RoboDK station: robodk_dot_following.rdk

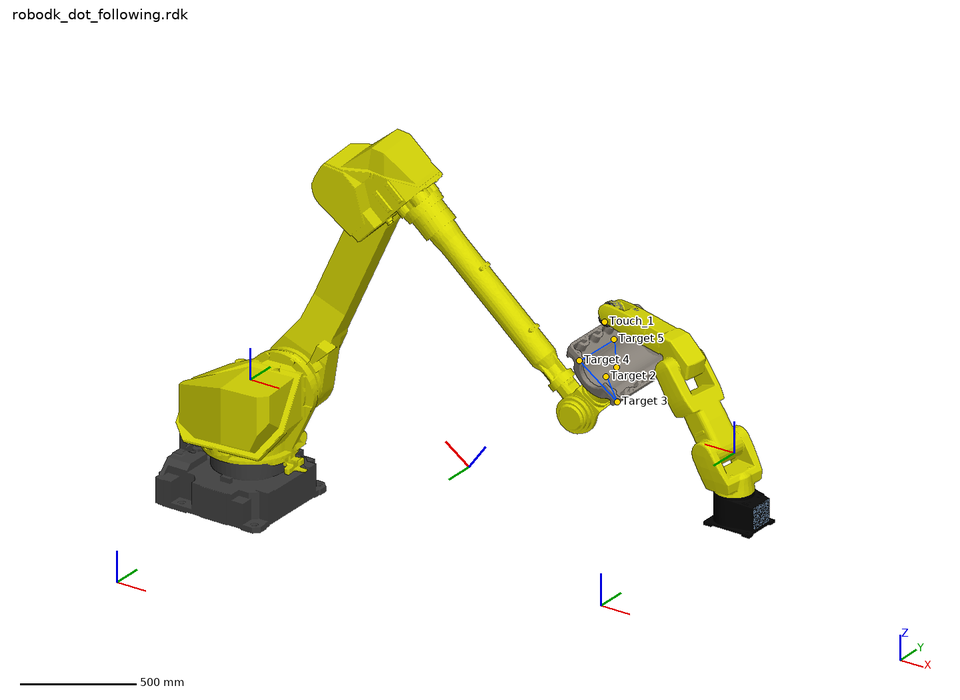
[picture v0: the station drawn from its stored meshes, robots at their saved joint values, targets as dots, program paths as lines]
Station Zavrsni_Beta (saved by RoboDK 5.9.4). Poses are relative to the parent item; angles as X-Y-Z fixed-axis rotations.
  - frame Pozicija 1 at (0, 0, 0) mm
    - frame Robot1 at (0, 1000, 570) mm
      - robot Robot1 (model Fanuc M-710iC/45M): 6 axes, payload 45 kg, reach 2606 mm, repeatability 0.06 mm, weight 570 kg
          modified DH rows (alpha deg, a mm, theta deg, d mm): 0, 0, 0, 570; -90, 150, -90, 0; 0, 1150, 0, 0; -90, 170, 0, 1295; 90, 0, 0, 0; -90, 0, 0, 175
          base shift (0, 0, -570) mm
          joint limits [-180, -110, -65, -360, -125, -360] to [180, 110, 245, 360, 125, 360]; home [0, 0, 0, 0, 0, 0]; saved at [4.644, 23.7, -43.76, -3.091, 98.158, 3.506]
        - tool OnRobot VGC10 Vacuum Gripper, TCP at (0, 0, 117.4) mm, size 100 x 100 x 114.9 mm
          - object Predmet at (-160, -250, 90) mm, size 330.2 x 509.8 x 126.9 mm, geometry from Part_Oil_Pan.sld
        - frame Frame 5 at (0, 1000, 0) mm
          - target Touch_1 (Cartesian target) at (158.88, -957.17, 281.93) mm, rotated rx -178.44 ry 2.6 rz 0.07 deg; joints [5.051, 6.745, -4.994, 9.729, -26.502, -11.335] of Robot2
    - target Target 2 (Cartesian target) at (1868.79, 1000, 1107.45) mm, rotated rx -1.55 ry -61.53 rz -180 deg; joints [0.282, 18.045, -39.644, -1.941, 68.13, 0.858] of Robot1
    - target Target 3 (Cartesian target) at (1925.5, 1000, 1002.89) mm, rotated rx -0.15 ry -61.53 rz -180 deg; joints [0.027, 23.437, -43.149, -0.184, 71.62, 0.071] of Robot1
    - target Target 4 (Cartesian target) at (1810.72, 881.58, 1214.55) mm, rotated rx 0 ry -61.53 rz 180 deg; joints [-4.359, 12.883, -35.614, 4.255, 64.216, -3.935] of Robot1
    - target Target 5 (Cartesian target) at (1815.88, 1134.09, 1217.34) mm, rotated rx 0 ry -61.53 rz -180 deg; joints [4.916, 13.107, -35.424, -4.806, 64.063, 4.454] of Robot1
    - target Target 7 (Cartesian target) at (1830.29, 1133.01, 1087.56) mm, rotated rx -0.23 ry -35.7 rz 179.79 deg; joints [4.644, 23.7, -43.76, -3.091, 98.158, 3.506] of Robot1
  - program Program_R1 (7 instructions, listed below)
  - frame Pozicija 2 at (2540, 0, 600) mm
    - frame Robot2 at (0, 1000, 330) mm, rotated rx 0 ry 0 rz -180 deg
      - robot Robot2: 6 axes
          modified DH rows (alpha deg, a mm, theta deg, d mm): 0, 0, 0, 330; -90, 75, -90, 0; 0, 400, 0, 0; -90, 75, 0, 410; 90, 0, 0, 0; -90, 0, 0, 80
          base shift (0, 0, -330) mm
          joint limits [-170, -60, -70, -190, -115, -400] to [170, 140, 170, 190, 115, 400]; home [0, 0, 0, 0, 0, 0]; saved at [-7.441, 35.58, 7.146, -5.827, -64.504, 8.653]
        - tool Robot2, TCP at (0, 0, 0) mm
  - Python program Dot_Following (listed below)
  - Python program Dot_Following_Record (listed below)
  - Python program Dot_Following_Replay (listed below)
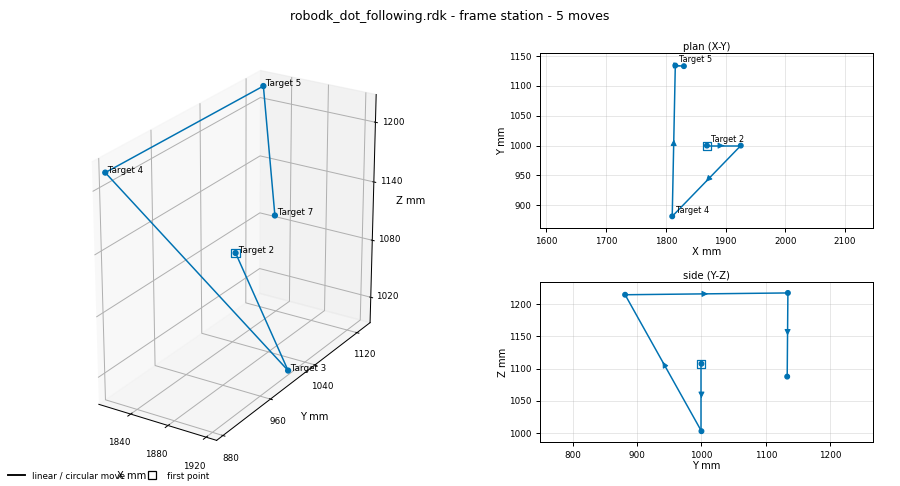
[picture p0: tool path of robodk_dot_following.rdk in frame station, 5 of 5 moves have a stored position in this frame; points joined in program order, loops and branches not executed]

--- program Program_R1 (robot Robot1) ---
  Set Ref.: Pozicija 1
  Set Tool: OnRobot VGC10 Vacuum Gripper
  MoveJ (Target 2)
  MoveL (Target 3)
  MoveL (Target 4)
  MoveL (Target 5)
  MoveL (Target 7)

--- Python program Dot_Following ---
from robodk.robolink import *
import time

RDK = Robolink()

robot2 = RDK.Item('Robot2', ITEM_TYPE_ROBOT)
touch  = RDK.Item('Touch_1', ITEM_TYPE_TARGET)
prog1  = RDK.Item('Program_R1', ITEM_TYPE_PROGRAM)

if not robot2.Valid(): raise Exception("Robot2 nije pronađen")
if not touch.Valid():  raise Exception("Touch_1 nije pronađen")
if not prog1.Valid():  raise Exception("Program_R1 nije pronađen")

# --- još malo brže (sigurno za simulaciju) ---
robot2.setSpeed(1200)          # mm/s
robot2.setAcceleration(5000)
robot2.setSpeedJoints(300)     # deg/s
robot2.setAccelerationJoints(900)

# 1) isto kao ručni klik
robot2.MoveJ(touch, blocking=True)

print("Robot2 na Touch_1. Pokrećem Robot1...")

# 2) pokreni Robot1
prog1.RunProgram()

print("Praćenje Touch_1 (200 Hz)")

# 3) HIGH-FREQ LOOP
DT = 0.005   # 200 Hz
t_next = time.time()

while prog1.Busy():
    now = time.time()
    if now < t_next:
        time.sleep(t_next - now)
    t_next += DT

    # non-stop "Go to Touch_1"
    robot2.MoveJ(touch, blocking=False)

print("Gotovo")

--- Python program Dot_Following_Record ---
from robodk.robolink import *
import time, csv
from datetime import datetime

RDK = Robolink()

robot1 = RDK.Item('Robot1', ITEM_TYPE_ROBOT)
robot2 = RDK.Item('Robot2', ITEM_TYPE_ROBOT)
touch  = RDK.Item('Touch_1', ITEM_TYPE_TARGET)
prog1  = RDK.Item('Program_R1', ITEM_TYPE_PROGRAM)

if not robot1.Valid(): raise Exception("Robot1 nije pronađen")
if not robot2.Valid(): raise Exception("Robot2 nije pronađen")
if not touch.Valid():  raise Exception("Touch_1 nije pronađen")
if not prog1.Valid():  raise Exception("Program_R1 nije pronađen")

DT = 0.005  # 200 Hz

# brzine (kao kod tebe)
robot2.setSpeed(1200)
robot2.setAcceleration(5000)
robot2.setSpeedJoints(300)
robot2.setAccelerationJoints(900)

stamp = datetime.now().strftime("%Y%m%d_%H%M%S")
CSV_FILE = rf"C:\Users\xgami\Desktop\R1R2_Record_{stamp}.csv"

# start Robot2 na Touch_1
robot2.MoveJ(touch, blocking=True)

# start Robot1 program
prog1.RunProgram()
print("RECORD start:", CSV_FILE)

t0 = time.time()
t_next = time.time()
n = 0

with open(CSV_FILE, "w", newline="") as f:
    w = csv.writer(f)
    # header: t + R1(6) + R2(6)
    w.writerow(["t",
                "R1_j1","R1_j2","R1_j3","R1_j4","R1_j5","R1_j6",
                "R2_j1","R2_j2","R2_j3","R2_j4","R2_j5","R2_j6"])

    while prog1.Busy():
        now = time.time()
        if now < t_next:
            time.sleep(t_next - now)
        t_next += DT

        # Robot2 prati Touch_1 (tvoj dokazano-radi način)
        robot2.MoveJ(touch, blocking=False)

        # snimi jointove oba robota
        j1 = robot1.Joints()
        j2 = robot2.Joints()

        j1_6 = [float(str(j1[i]).replace('[','').replace(']','').strip()) for i in range(6)]
        j2_6 = [float(str(j2[i]).replace('[','').replace(']','').strip()) for i in range(6)]

        w.writerow([time.time()-t0] + j1_6 + j2_6)
        n += 1

print("RECORD gotov. Uzoraka:", n)
print("Spremljeno u:", CSV_FILE)

--- Python program Dot_Following_Replay ---
from robodk.robolink import *
import time, csv, glob, os

RDK = Robolink()

robot1 = RDK.Item('Robot1', ITEM_TYPE_ROBOT)
robot2 = RDK.Item('Robot2', ITEM_TYPE_ROBOT)

if not robot1.Valid(): raise Exception("Robot1 nije pronađen")
if not robot2.Valid(): raise Exception("Robot2 nije pronađen")

# najnoviji record
pattern = r"C:\Users\xgami\Desktop\R1R2_Record_*.csv"
files = glob.glob(pattern)
if not files:
    raise Exception(f"Nema fileova: {pattern}")

CSV_FILE = max(files, key=os.path.getmtime)
print("Koristim file:", CSV_FILE)

def to_float(x):
    s = str(x).replace('[','').replace(']','').strip()
    return float(s)

# učitaj
data = []
with open(CSV_FILE, newline="") as f:
    r = csv.reader(f)
    next(r, None)
    for row in r:
        if not row:
            continue
        vals = [to_float(x) for x in row[:13]]  # t + 12 jointova
        data.append(vals)

if len(data) < 2:
    raise Exception("CSV prekratak")

print("REPLAY start (R1 + R2)")

t_start = time.time()
for row in data:
    t = row[0]
    r1 = row[1:7]
    r2 = row[7:13]

    while (time.time() - t_start) < t:
        time.sleep(0.0005)

    robot1.setJoints(r1)
    robot2.setJoints(r2)

print("REPLAY gotov.")
